{attribute 'qualified_only'}
VAR_GLOBAL
	Axis1 : AXIS_REF;
	Axis2 : AXIS_REF;
END_VAR

(* stored: Version 1.1.0.1
   GVL GVL_Axes: Id {c8a64daa-ce3e-4d1a-97fd-9b8ae50d2992} *)
